Staubli VAL3: root.pgx

public program root(num& x_nInput[], num& x_nResult[])
  local num l_nLength
  local num l_nElement
begin

  l_nLength = size(x_nInput)
  resize(x_nResult,1,1)
  x_nResult = 0
  resize(x_nResult,1,l_nLength)

  for l_nElement = 0 to l_nLength -1
    x_nResult[l_nElement] = power(x_nInput[l_nElement],0.5)
  endFor

end
